// TIA Portal V18 export
// export: Created 2026-06-08T16:32:21.6821168Z, ExportSetting WithDefaults, DisplayName Totally Integrated Automation Portal, DisplayVersion V18, DisplayName TIA Portal Openness, DisplayVersion V18, DisplayName TIA Portal Version Control Interface, DisplayVersion V18, DisplayName STEP 7 Professional, DisplayVersion V18, DisplayName STEP 7 Safety, DisplayVersion V18, DisplayName WinCC Professional, DisplayVersion V18
DATA_BLOCK "Assembly_Emergency_DB_1"   // DB34
VERSION : 0.1
// stored: AutoNumber true, InstanceOfName Assembly_Emergency, InstanceOfType FB
"Assembly_Emergency"
BEGIN
END_DATA_BLOCK
